(* IEC 61131-3 sources: verifaps-lib/run/src/test/resources/edu/kit/iti/formal/automation/run, 13 files *)

(* ---- runtimeTest.functionBlockTest.st ---- *)
FUNCTION_BLOCK TON

VAR_INPUT
    IN : BOOL;
    IN2 : BOOL;
END_VAR

VAR_OUTPUT
    Q  : BOOL := TRUE;
END_VAR

    Q := IN AND IN2;

END_FUNCTION_BLOCK

PROGRAM  Analogsensor

    VAR
      timeout          	: TON;
      e : BOOL;
    END_VAR

    timeout(IN := TRUE, IN2 := TRUE);

    e := timeout.Q;

END_PROGRAM

(* ---- expressionVisitorTest.basicTest.st ---- *)
TYPE
    MY_ENUM : (possible, values, enum);
END_TYPE

PROGRAM my_sth
    VAR_INPUT
        active : BOOL := True;
        number : INT := 1;
        my_enum : MY_ENUM;
    END_VAR

    VAR_OUTPUT
        my_output : MY_ENUM;
        seriously : BOOL;
    END_VAR

    VAR
        my_enum_local : MY_ENUM;
    END_VAR

    VAR_IN_OUT
        active_inout : BOOL;
    END_VAR

   seriously := NOT FALSE;
   number := (- 19);
   number := 1 + 2;

END_PROGRAM

(* ---- runtimeTest.advancedTest.st ---- *)
TYPE
    TrafficLight : (Red, Green);
END_TYPE

PROGRAM PedestrianTrafficLight

    VAR_INPUT
        pedBtnPress : BOOL := true;
    END_VAR

    VAR_OUTPUT
        carLight : TrafficLight;
        pedLight : TrafficLight;
        counter : INT := 50;
    END_VAR

    VAR
        buttonPressedBefore : BOOL := false;
    END_VAR

    IF (NOT buttonPressedBefore) AND pedBtnPress THEN
        carLight := TrafficLight#Red;
    END_IF

    IF counter = 10 THEN
        pedLight := TrafficLight#Green;
    ELSIF counter = 40 THEN
     pedLight := TrafficLight#Red;
    ELSIF counter = 50 THEN
        carLight := TrafficLight#Green;
    END_IF

    IF carLight = TrafficLight#Red THEN
        counter := counter + 1;
    ELSE
        counter := 0;
    END_IF

    buttonPressedBefore := pedBtnPress;

END_PROGRAM

(* ---- runtimeTest.cycles.st ---- *)
PROGRAM my_sth
    VAR_INPUT
        I : INT;
    END_VAR

    VAR
        counter : INT := 0;
    END_VAR

   counter := counter + I;

   IF counter > 1000 THEN
        counter := 0;
   END_IF

END_PROGRAM

(* ---- runtimeTest.elevatorTest.st ---- *)
TYPE
  MOTOR_STATE : (GoDown, Stationary, GoUp);
  DOOR_STATE : (Open, Closed);
END_TYPE

PROGRAM Elevator

  VAR_INPUT
    CurrentPos : INT := 3;
    RequestedPos : INT := 5;
    ButtonPressed : BOOL;
  END_VAR

  VAR_OUTPUT
    Motor : MOTOR_STATE := MOTOR_STATE#Stationary;
    Door : DOOR_STATE := DOOR_STATE#Open;
  END_VAR

  IF ButtonPressed THEN

    Door := DOOR_STATE#Closed;

    IF RequestedPos > CurrentPos THEN
      Motor := MOTOR_STATE#GoUp;
    ELSEIF RequestedPos < CurrentPos THEN
      Motor := MOTOR_STATE#GoDown;
    END_IF

  END_IF

  IF RequestedPos = CurrentPos THEN
    Motor := MOTOR_STATE#Stationary;
    Door := DOOR_STATE#Open;
  END_IF

END_PROGRAM

(* ---- runtimeTest.enumTest.st ---- *)
TYPE
    MY_ENUM : (possible, values, enum);
END_TYPE

PROGRAM my_sth
    VAR_INPUT
        active : BOOL := True;
        number : INT := 1;
        my_enum : MY_ENUM;
    END_VAR

   seriously := NOT FALSE;
   number := (- 19);
   number := number + 2;
   seriously := NOT seriously;
   number := 3;

   if number = 3 THEN
    number :=300;
   END_IF
END_PROGRAM

(* ---- runtimeTest.forLoopTest.st ---- *)
PROGRAM my_sth
    VAR_INPUT
        Var1 : INT := 2;
        Var2 : INT := 0;
        counter2 : INT := 0;
    END_VAR

   FOR counter:=1 TO 5 BY 1 DO
       Var1:=Var1*2;
   END_FOR

   FOR counter2:=1 TO 5 BY 1 DO
      Var2:=Var2+1;
      counter2:=counter2+3;
   END_FOR
END_PROGRAM

(* ---- runtimeTest.functionTest.st ---- *)
FUNCTION FuncAdd : REAL
VAR_INPUT
    a: REAL;
    b: REAL;
END_VAR

FuncAdd := 2*a - 22*b;
END_FUNCTION

PROGRAM my_sth
    VAR_INPUT
        Var1 : REAL := 2;
        x : REAL := 7;
        y : REAL := 8;
    END_VAR

   Var1 := FuncAdd(x, y);
END_PROGRAM

(* ---- runtimeTest.repeatLoopTest.st ---- *)
PROGRAM my_sth
    VAR_INPUT
        Var1 : INT := 2;
        counter : INT := 4;
    END_VAR

   REPEAT
       Var1 := Var1*2;
       counter := counter-1;
   UNTIL
       counter=0
   END_REPEAT
END_PROGRAM

(* ---- runtimeTest.structTest.st ---- *)
TYPE Point: STRUCT
                x: INT; y: INT;
            END_STRUCT;
END_TYPE

PROGRAM my_sth
    VAR
        Var1 : Point;
        Var2 : INT;
        Var3 : Point := (x:= 1, y:=2);
    END_VAR

    Var2 := 7;
    Var1.x := 1;
    Var1.y := 2;
    Var3.y := 100;
    Var3.y := -70000;

END_PROGRAM

(* ---- runtimeTest.testIfStatement.st ---- *)
PROGRAM my_sth
    VAR_INPUT
        number : INT := 1;
        n2 : INT;
        active : BOOL := True;
    END_VAR

   number := 3;

   if number = 3 THEN
    number :=300;
   END_IF

   if active THEN
    n2 := 4;
    END_IF
END_PROGRAM

(* ---- runtimeTest.testVariableReference.st ---- *)
PROGRAM my_sth
    VAR_INPUT
        b : BOOL := True;
        b2 : BOOL;
        number : INT := 1;
        n2 : INT;
        n3 : INT := 4;
        n4 : INT;
        n5 : INT := 3;
        n6 : INT := 13;
        n7 : INT := 3;
        n8, n9, n10 : BOOL;
    END_VAR

    b2 := NOT FALSE;
    number := (- 19);
    n2 := (- 3)+ 2;
    b := NOT b;
    n5 := n5 * 2;
    n6 := n6 MOD 7;
    n7 := n7 - 4;
    n8 := 3 <> 4;
    n9 := 3 < 4 AND 3 <= 3 AND -4 < 5 AND 4 <= 7;
    n10 := 4 < 3 OR 4 <= 3 OR 6 < -5;
END_PROGRAM

(* ---- runtimeTest.whileLoopTest.st ---- *)
PROGRAM my_sth
    VAR_INPUT
        Var1 : INT := 2;
        counter : INT := 4;
    END_VAR

   WHILE counter<>0 DO
       Var1 := Var1*2;
       counter := counter-1;
   END_WHILE
END_PROGRAM
